DATA_BLOCK "IAI_Position_DB"
{ S7_Optimized_Access := 'TRUE' }
VERSION : 0.1
NON_RETAIN
"IAI_Position"

BEGIN

END_DATA_BLOCK

